/// configuration data that is used during boot to configure the Units equipment
TYPE MoverDataConfig :
STRUCT
  Simulated : BOOL;
END_STRUCT
END_TYPE

(* stored: Version 1.1.0.1
   DUT MoverDataConfig: Id {eedda42a-aeda-4e01-b60e-934ee44ab470} *)
